TYPE TFMachineTransport_GatesAccess :
STRUCT
		
	GateAccessCarico 			: TFGateAccess;
	GateAccessCentratoreEsterno	: TFGateAccess;
	
END_STRUCT
END_TYPE

(* stored: Version 1.1.0.1, ProductVersion 3.1.4024.11
   DUT TFMachineTransport_GatesAccess: Id {7ba4761b-e085-4404-b183-8fb81a34d804} *)
